(* LS Electric XG5000 project: 241007_펑션 실습1 *)
(* PLC LSPLC *)
(* module base 0 slot 0: 입력 모듈:XGI-D22A/B (DC 24V 입력, 16점 (전류소스 싱크공용/ 전류소스 입력)) *)
(* module base 0 slot 1: 출력 모듈:XGQ-RY2A/B (릴레이 출력, 16점 (2A용, Varistor 없음/Varistor 부착)) *)

PROGRAM NewProgram (* task: 스캔 프로그램 *)
VAR
    결과 : REAL;
    결과1 : REAL;
    결과2 : INT;
    숫자1 : INT := 10;
END_VAR

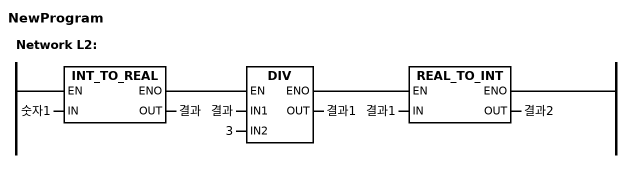
(* Rung L2 *)
결과 := INT_TO_REAL(숫자1);
결과1 := 결과 / 3;
결과2 := REAL_TO_INT(결과1);
END_PROGRAM